// Core §3.8 local provider. Validation is generic BECAUSE SchemaVersion is the
// first UINT of every ParCfg/record (§3.8): stored first-UINT must equal the
// target's initialized first-UINT, else Load = FALSE and the caller faults
// RECIPE_INVALID. Never a partial apply. Types stage through PrepareRecipe.
FUNCTION_BLOCK FB_LocalRecipeProvider IMPLEMENTS I_RecipeProvider, I_RecipeStore
VAR
    _n    : INT;
    _models : ARRAY[1..PL_Fraktal.MAX_RECIPES] OF STRING(80);
    _keys   : ARRAY[1..PL_Fraktal.MAX_RECIPES] OF STRING(80);
    {attribute 'OPC.UA.DA' := '0'}
    _ptr  : ARRAY[1..PL_Fraktal.MAX_RECIPES] OF PVOID;
    _size : ARRAY[1..PL_Fraktal.MAX_RECIPES] OF UDINT;
END_VAR

// no cyclic body

METHOD Load : BOOL
VAR_INPUT
    ModelCode : STRING;
    RecipeKey : STRING;
    pParCfg : PVOID;
    Size    : UDINT;
END_VAR
VAR
    i, hit, fallback : INT;
    puT, puS : POINTER TO UINT;
END_VAR
Load := FALSE;
hit := 0;
fallback := 0;
FOR i := 1 TO _n DO
    IF (_keys[i] = RecipeKey) AND (_models[i] = ModelCode) THEN
        hit := i;
        EXIT;
    ELSIF (_keys[i] = RecipeKey) AND (_models[i] = '') THEN
        fallback := i;
    END_IF
END_FOR
IF hit = 0 THEN
    hit := fallback;
END_IF
// Two statements, not one condition: IEC 61131-3 does not mandate short-circuit
// evaluation and TwinCAT's compile option for it is off by default, so a single
// `(hit = 0) OR (_size[hit] <> Size)` still reads _size[0] on the ordinary
// not-found path - out of bounds for ARRAY[1..MAX_RECIPES] (§3.8).
IF (hit = 0) OR (pParCfg = 0) THEN
    RETURN;                                       // unknown recipe -> caller faults (§3.8)
END_IF
IF _size[hit] <> Size THEN
    RETURN;                                       // size mismatch -> caller faults (§3.8)
END_IF
puT := pParCfg;
puS := _ptr[hit];
IF puT^ <> puS^ THEN
    RETURN;                                       // SchemaVersion mismatch: migrate-or-fault (§3.8)
END_IF
MEMCPY(destAddr := pParCfg, srcAddr := _ptr[hit], n := Size);
Load := TRUE;
END_METHOD

// I_RecipeStore - write an edited record back into the registered storage of
// exactly (ModelCode, RecipeKey). The fallback record is never edited in a
// specific model's name, and a size or SchemaVersion mismatch changes nothing.
METHOD Save : BOOL
VAR_INPUT
    ModelCode : STRING;
    RecipeKey : STRING;
    pData     : PVOID;
    Size      : UDINT;
END_VAR
VAR
    i, hit : INT;
    puT, puS : POINTER TO UINT;
END_VAR
Save := FALSE;
hit := 0;
FOR i := 1 TO _n DO
    IF (_keys[i] = RecipeKey) AND (_models[i] = ModelCode) THEN
        hit := i;
        EXIT;
    END_IF
END_FOR
IF (hit = 0) OR (pData = 0) THEN
    RETURN;
END_IF
IF _size[hit] <> Size THEN
    RETURN;
END_IF
puT := _ptr[hit];
puS := pData;
IF puT^ <> puS^ THEN
    RETURN;                                       // SchemaVersion differs: nothing written
END_IF
MEMCPY(destAddr := _ptr[hit], srcAddr := pData, n := Size);
Save := TRUE;
END_METHOD

// application wiring: one record per (ModelCode, RecipeKey); empty ModelCode is fallback.
METHOD Register : BOOL
VAR_INPUT
    ModelCode : STRING(80);
    RecipeKey : STRING(80);
    pData  : PVOID;
    Size   : UDINT;
END_VAR
VAR
    i : INT;
END_VAR
IF (_n >= PL_Fraktal.MAX_RECIPES) OR (pData = 0) OR (RecipeKey = '') THEN
    Register := FALSE;
    RETURN;
END_IF
FOR i := 1 TO _n DO
    IF (_models[i] = ModelCode) AND (_keys[i] = RecipeKey) THEN
        Register := FALSE;
        RETURN;
    END_IF
END_FOR
_n := _n + 1;
_models[_n] := ModelCode;
_keys[_n]   := RecipeKey;
_ptr[_n]  := pData;
_size[_n] := Size;
Register := TRUE;
END_METHOD

PROPERTY Ready : BOOL
GET
Ready := (_n > 0);
END_GET
END_PROPERTY

PROPERTY Source : E_RecipeSource
GET
Source := E_RecipeSource.LOCAL;
END_GET
END_PROPERTY

END_FUNCTION_BLOCK

(* stored: Version 1.1.0.1, ProductVersion 3.1.4024.12
   POU FB_LocalRecipeProvider: Id {1c0f8ef1-f5d0-4936-be06-851daa076225}, SpecialFunc None
   Method Load: Id {b1aef472-8321-4e67-becf-11964cf574b7}
   Method Save: Id {94fd026d-2726-4a9c-be43-91276ef36e97}
   Method Register: Id {df7be18b-5d33-4de5-8a36-02fc90bfd518}
   Property Ready: Id {5012cd35-f8d3-4752-893d-710a9a976af9}
   Get Get: Id {ed439f68-57a6-4ba8-9c56-d5b8a2eb482c}
   Property Source: Id {f8bb7684-b985-4251-a2ed-a6cff3c51e9c}
   Get Get: Id {702d2ac1-64c4-4474-8c33-95a6f866cc73} *)
